// TIA Portal project "TIA Add-in Testing" (V16)

(* hardware
DEVICE "stationMain"  S7-1500 station
   slot 0: "Rail_0"  Rack  6ES7 590-1***0-0AA0
   slot 1: "Main"  CPU 1516-3 PN/DP  6ES7 516-3AN01-0AB0  V2.8
      slot 3: "CPU display_1"  6ES7591-1BA00-0AA0
      slot 32768: "PROFINET interface_1"  X1
         slot 32769: "Port_1"  X1 P1
         slot 32770: "Port_2"  X1 P2
      slot 33024: "PROFINET interface_2"  X2
         slot 33025: "Port_1"  X2 P1
      slot 33280: "DP interface_1"  X3
      slot 34817: "Virtual CP interface port_1"  Virtual CP interface port  Virtual CP interface port
DEVICE "stationPlant"  S7-1500 station
   slot 0: "Rail_0"  Rack  6ES7 590-1***0-0AA0
   slot 1: "Plant"  CPU 1516-3 PN/DP  6ES7 516-3AN01-0AB0  V2.8
      slot 3: "CPU display_1"  6ES7591-1BA00-0AA0
      slot 32768: "PROFINET interface_1"  X1
         slot 32769: "Port_1"  X1 P1
         slot 32770: "Port_2"  X1 P2
      slot 33024: "PROFINET interface_2"  X2
         slot 33025: "Port_1"  X2 P1
      slot 33280: "DP interface_1"  X3
      slot 34817: "Virtual CP interface port_1"  Virtual CP interface port  Virtual CP interface port
DEVICE "stationLine"  S7-1500 station
   slot 0: "Rail_0"  Rack  6ES7 590-1***0-0AA0
   slot 1: "Line"  CPU 1516-3 PN/DP  6ES7 516-3AN01-0AB0  V2.8
      slot 3: "CPU display_1"  6ES7591-1BA00-0AA0
      slot 32768: "PROFINET interface_1"  X1
         slot 32769: "Port_1"  X1 P1
         slot 32770: "Port_2"  X1 P2
      slot 33024: "PROFINET interface_2"  X2
         slot 33025: "Port_1"  X2 P1
      slot 33280: "DP interface_1"  X3
      slot 34817: "Virtual CP interface port_1"  Virtual CP interface port  Virtual CP interface port
DEVICE "stationrack1"  ET 200SP-Station
   slot 0: "Rack_0"  Rack  6ES5 710-8MAx1
   slot 0: "rack1"  IM 155-6 PN ST  6ES7 155-6AU01-0BN0  V4.1
   slot 1: "DI1"  DI 8x24VDC ST  6ES7 131-6BF01-0BA0  V0.0
      slot 1: "DI1"  DI 8x24VDC ST
   slot 2: "DO2"  DQ 8x24VDC/0.5A ST  6ES7 132-6BF01-0BA0  V0.0
      slot 1: "DO2"  DQ 8x24VDC/0.5A ST
   slot 3: "AI3"  AI 2xU/I 2-,4-wire HF  6ES7 134-6HB00-0CA1  V2.0
      slot 1: "AI3"  AI 2xU/I 2-,4-wire HF
   slot 4: "AO4"  AQ 4xU/I ST  6ES7 135-6HD00-0BA1  V1.1
      slot 1: "AO4"  AQ 4xU/I ST
   slot 5: "Server module_1"  Server module  6ES7 193-6PA00-0AA0  V1.1
      slot 1: "Server module_1"  Server module
   slot 127: "BA 2xRJ45"  BA 2xRJ45  6ES7 193-6AR00-0AA0  V0.0
      slot 1: "Port_1"  X1 P1 R  6ES7 193-6AR00-0AA0  V0.0
      slot 2: "Port_2"  X1 P2 R  6ES7 193-6AR00-0AA0  V0.0
DEVICE "stationrack2"  ET 200SP-Station
   slot 0: "Rack_0"  Rack  6ES5 710-8MAx1
   slot 0: "rack2"  IM 155-6 PN ST  6ES7 155-6AU01-0BN0  V4.1
   slot 1: "DI1"  DI 8x24VDC ST  6ES7 131-6BF01-0BA0  V0.0
      slot 1: "DI1"  DI 8x24VDC ST
   slot 2: "DO2"  DQ 8x24VDC/0.5A ST  6ES7 132-6BF01-0BA0  V0.0
      slot 1: "DO2"  DQ 8x24VDC/0.5A ST
   slot 3: "AI3"  AI 2xU/I 2-,4-wire HF  6ES7 134-6HB00-0CA1  V2.0
      slot 1: "AI3"  AI 2xU/I 2-,4-wire HF
   slot 4: "AO4"  AQ 4xU/I ST  6ES7 135-6HD00-0BA1  V1.1
      slot 1: "AO4"  AQ 4xU/I ST
   slot 5: "Server module_1"  Server module  6ES7 193-6PA00-0AA0  V1.1
      slot 1: "Server module_1"  Server module
   slot 127: "BA 2xRJ45"  BA 2xRJ45  6ES7 193-6AR00-0AA0  V0.0
      slot 1: "Port_1"  X1 P1 R  6ES7 193-6AR00-0AA0  V0.0
      slot 2: "Port_2"  X1 P2 R  6ES7 193-6AR00-0AA0  V0.0
DEVICE "stationrack3"  ET 200SP-Station
   slot 0: "Rack_0"  Rack  6ES5 710-8MAx1
   slot 0: "rack3"  IM 155-6 PN ST  6ES7 155-6AU01-0BN0  V4.1
   slot 1: "DI1"  DI 8x24VDC ST  6ES7 131-6BF01-0BA0  V0.0
      slot 1: "DI1"  DI 8x24VDC ST
   slot 2: "DO2"  DQ 8x24VDC/0.5A ST  6ES7 132-6BF01-0BA0  V0.0
      slot 1: "DO2"  DQ 8x24VDC/0.5A ST
   slot 3: "AI3"  AI 2xU/I 2-,4-wire HF  6ES7 134-6HB00-0CA1  V2.0
      slot 1: "AI3"  AI 2xU/I 2-,4-wire HF
   slot 4: "AO4"  AQ 4xU/I ST  6ES7 135-6HD00-0BA1  V1.1
      slot 1: "AO4"  AQ 4xU/I ST
   slot 5: "Server module_1"  Server module  6ES7 193-6PA00-0AA0  V1.1
      slot 1: "Server module_1"  Server module
   slot 127: "BA 2xRJ45"  BA 2xRJ45  6ES7 193-6AR00-0AA0  V0.0
      slot 1: "Port_1"  X1 P1 R  6ES7 193-6AR00-0AA0  V0.0
      slot 2: "Port_2"  X1 P2 R  6ES7 193-6AR00-0AA0  V0.0
DEVICE "stationrack4"  ET 200SP-Station
   slot 0: "Rack_0"  Rack  6ES5 710-8MAx1
   slot 0: "rack4"  IM 155-6 PN ST  6ES7 155-6AU01-0BN0  V4.1
   slot 1: "DI1"  DI 8x24VDC ST  6ES7 131-6BF01-0BA0  V0.0
      slot 1: "DI1"  DI 8x24VDC ST
   slot 2: "DO2"  DQ 8x24VDC/0.5A ST  6ES7 132-6BF01-0BA0  V0.0
      slot 1: "DO2"  DQ 8x24VDC/0.5A ST
   slot 3: "AI3"  AI 2xU/I 2-,4-wire HF  6ES7 134-6HB00-0CA1  V2.0
      slot 1: "AI3"  AI 2xU/I 2-,4-wire HF
   slot 4: "AO4"  AQ 4xU/I ST  6ES7 135-6HD00-0BA1  V1.1
      slot 1: "AO4"  AQ 4xU/I ST
   slot 5: "Server module_1"  Server module  6ES7 193-6PA00-0AA0  V1.1
      slot 1: "Server module_1"  Server module
   slot 127: "BA 2xRJ45"  BA 2xRJ45  6ES7 193-6AR00-0AA0  V0.0
      slot 1: "Port_1"  X1 P1 R  6ES7 193-6AR00-0AA0  V0.0
      slot 2: "Port_2"  X1 P2 R  6ES7 193-6AR00-0AA0  V0.0
DEVICE "stationrack5"  ET 200SP-Station
   slot 0: "Rack_0"  Rack  6ES5 710-8MAx1
   slot 0: "rack5"  IM 155-6 PN ST  6ES7 155-6AU01-0BN0  V4.1
   slot 1: "DI1"  DI 8x24VDC ST  6ES7 131-6BF01-0BA0  V0.0
      slot 1: "DI1"  DI 8x24VDC ST
   slot 2: "DO2"  DQ 8x24VDC/0.5A ST  6ES7 132-6BF01-0BA0  V0.0
      slot 1: "DO2"  DQ 8x24VDC/0.5A ST
   slot 3: "AI3"  AI 2xU/I 2-,4-wire HF  6ES7 134-6HB00-0CA1  V2.0
      slot 1: "AI3"  AI 2xU/I 2-,4-wire HF
   slot 4: "AO4"  AQ 4xU/I ST  6ES7 135-6HD00-0BA1  V1.1
      slot 1: "AO4"  AQ 4xU/I ST
   slot 5: "Server module_1"  Server module  6ES7 193-6PA00-0AA0  V1.1
      slot 1: "Server module_1"  Server module
   slot 127: "BA 2xRJ45"  BA 2xRJ45  6ES7 193-6AR00-0AA0  V0.0
      slot 1: "Port_1"  X1 P1 R  6ES7 193-6AR00-0AA0  V0.0
      slot 2: "Port_2"  X1 P2 R  6ES7 193-6AR00-0AA0  V0.0
*)

// ===== PLC "Main"  CPU 1516-3 PN/DP =====

VAR_GLOBAL   // PLC tag table "autoGenTags"
   "Digital Input 1" AT %I0.0 : Bool;
   "Door Open" AT %I0.1 : Bool;
   "Door Close" AT %I0.2 : Bool;
   "Limit Switch" AT %I0.3 : Bool;
   "Digital Output 1" AT %Q0.0 : Bool;
   "Analog Input" AT %IW1 : Word;
   "Analog Output" AT %QW1 : Word;
   "Digital Input 2" AT %I5.0 : Bool;
   "Digital Output 2" AT %Q9.0 : Bool;
   "Analog Input 2" AT %IW6 : Word;
   "Analog Output 2" AT %QW10 : Word;
   "Digital Input 3" AT %I10.0 : Bool;
   "Digital Output 3" AT %Q18.0 : Bool;
   "Analog Input 3" AT %IW11 : Word;
   "Analog Output 3" AT %QW19 : Word;
END_VAR

ORGANIZATION_BLOCK "Main"   // OB1, LAD, ProgramCycle
TITLE = "Main Program Sweep (Cycle)"
{ S7_Optimized_Access := 'TRUE' }
VERSION : 0.1
   VAR_INPUT
      Initial_Call : Bool;   // Initial call of this OB
      Remanence : Bool;   // =True, if remanent data are available
   END_VAR
BEGIN
END_ORGANIZATION_BLOCK

// ===== PLC "Plant"  CPU 1516-3 PN/DP =====

VAR_GLOBAL   // PLC tag table "autoGenTags"
   "Digital Input 1" AT %I0.0 : Bool;
   "Digital Output 1" AT %Q0.0 : Bool;
   "Analog Input" AT %IW1 : Word;
   "Analog Output" AT %QW1 : Word;
END_VAR

ORGANIZATION_BLOCK "Main"   // OB1, LAD, ProgramCycle
TITLE = "Main Program Sweep (Cycle)"
{ S7_Optimized_Access := 'TRUE' }
VERSION : 0.1
   VAR_INPUT
      Initial_Call : Bool;   // Initial call of this OB
      Remanence : Bool;   // =True, if remanent data are available
   END_VAR
BEGIN
END_ORGANIZATION_BLOCK

// ===== PLC "Line"  CPU 1516-3 PN/DP =====

VAR_GLOBAL   // PLC tag table "autoGenTags"
   "Digital Input 1" AT %I0.0 : Bool;
   "Digital Output 1" AT %Q0.0 : Bool;
   "Analog Input" AT %IW1 : Word;
   "Analog Output" AT %QW1 : Word;
END_VAR

ORGANIZATION_BLOCK "Main"   // OB1, LAD, ProgramCycle
TITLE = "Main Program Sweep (Cycle)"
{ S7_Optimized_Access := 'TRUE' }
VERSION : 0.1
   VAR_INPUT
      Initial_Call : Bool;   // Initial call of this OB
      Remanence : Bool;   // =True, if remanent data are available
   END_VAR
BEGIN
END_ORGANIZATION_BLOCK